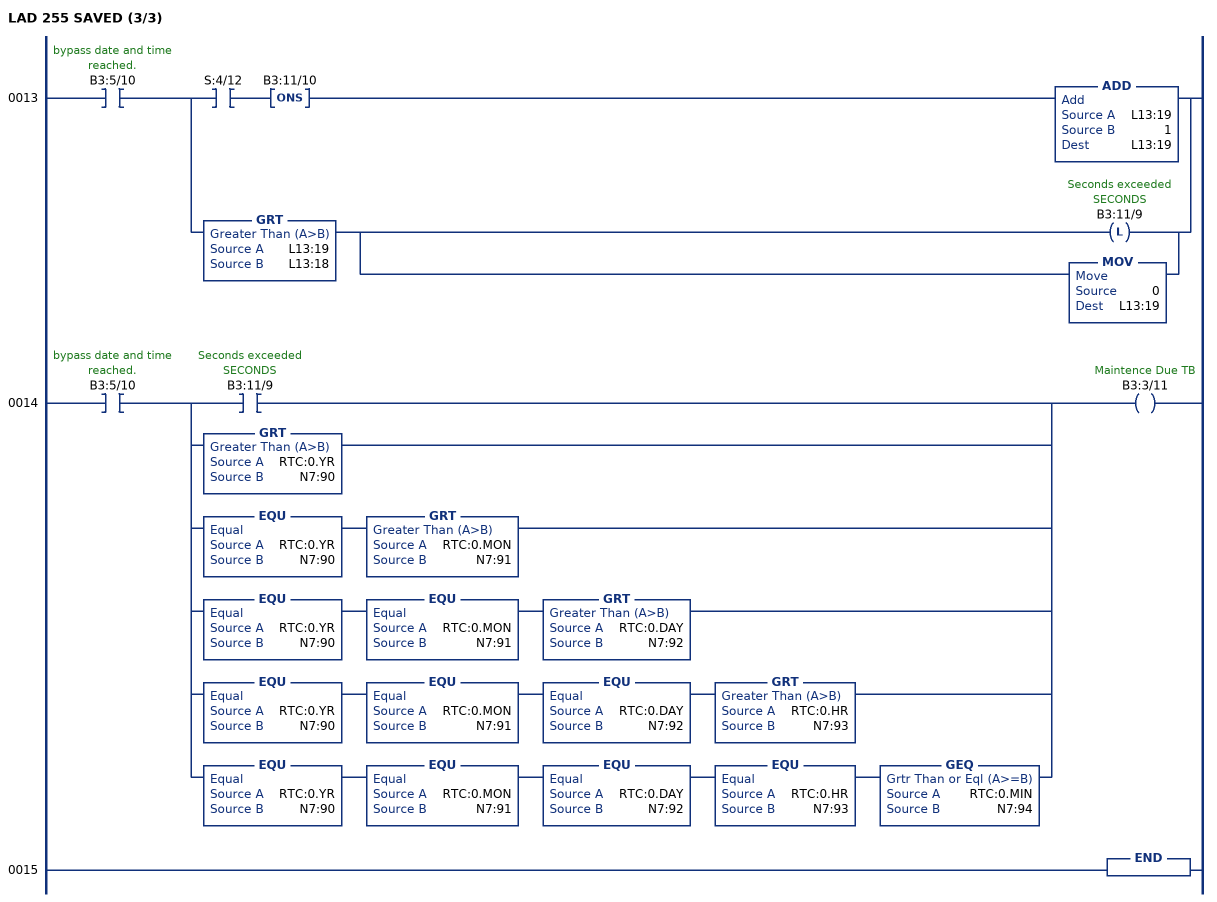
% Rung: 13 %
SOR XIC B3:5/10 BST XIC S:4/12 ONS B3:11/10 ADD L13:19 1 L13:19 NXB GRT L13:19 L13:18 BST OTL B3:11/9 NXB MOV 0 L13:19 BND BND EOR
%   B3:5/10  "bypass date and time reached." %
%   L13:18  MAX %
%   B3:11/9  SECONDS  "Seconds exceeded" %
% Rung: 14 %
SOR XIC B3:5/10 BST XIC B3:11/9 NXB GRT RTC:0.YR N7:90 NXB EQU RTC:0.YR N7:90 GRT RTC:0.MON N7:91 NXB EQU RTC:0.YR N7:90 EQU RTC:0.MON N7:91 GRT RTC:0.DAY N7:92 NXB EQU RTC:0.YR N7:90 EQU RTC:0.MON N7:91 EQU RTC:0.DAY N7:92 GRT RTC:0.HR N7:93 NXB EQU RTC:0.YR N7:90 EQU RTC:0.MON N7:91 EQU RTC:0.DAY N7:92 EQU RTC:0.HR N7:93 GEQ RTC:0.MIN N7:94 BND OTE B3:3/11 EOR
%   B3:5/10  "bypass date and time reached." %
%   B3:11/9  SECONDS  "Seconds exceeded" %
%   N7:90  RTC %
%   B3:3/11  TB  "Maintence Due" %
% Rung: 15 %
SOR END EOR

OTHER DOCUMENTED ADDRESSES
  B3:0/1  "toggle"
  B3:0/13  "toggle 2"
  B3:10/1  "bypass"
  B189:0/0  "change box"
  B189:0/9  "override boxing ok or not full signal"
  B189:0/11  "HMI force door close"
  B196:1/0  "Chute door is closed"
  B196:1/1  "control chute door"
  B196:1/13  "force box conveyor on"
  B196:3/0  "for hmi to continue production unlatched by hmi"
  HSC:0.0  "top"
  HSC:0.3/6  "Underflow interrupt"
  HSC:0.3/7  "Overflow interrupt"
  HSC:1.0  "bot"
  HSC:1.3/6  "Underflow interrupt"
  HSC:1.3/7  "Overflow interrupt"
  I:0.0/0  "Encoder Signal "A""
  I:0.0/1  "Encoder Signal "B""
  I:0.0/4  "Encoder Signal "A""
  I:0.0/5  "Encoder Signal "B""
  I:0.1/4  "not used"
  I:0.1/5  "not used"
  I:0.1/6  "not used"
  I:0.1/7  "not used"
  I:0.1/8  "not used"
  I:0.1/9  "not used"
  I:0.1/10  "not used"
  I:0.1/11  "not used"
  I:0.1/12  "not used"
  I:0.1/13  "not used"
  I:0.1/14  "not used"
  I:0.1/15  "not used"
  I:0.2  "not used"
  I:0.2/3  "Packaging Conveyor full"
  I:0.2/4  "Packaging Conveyor Box in Position"
  I:0.3  "not used"
  I:0.4  "Spare Analog Input 1"
  I:0.5  "Spare Analog Input 2"
  I:0.6  "Spare Analog Input 3"
  I:2.0/0  FRONT_ESTOP
  I:2.0/1  REAR_ESTOP
  I:2.0/8  FRONT_DOOR  "front door signal ce models only"
  I:2.0/9  REAR_DOOR  "rear door signal ce models only"
  I:2.0/11  "spare"
  L23:19  TOP_OPT_FAIL_CT
  L23:34  AIR_PRESSURE_FAULT
  L28:0  INS_1_TIME
  L29:0  INS_1_POS
  L30:0  INS_5_TIME
  L31:0  INS_5_POS
  L32:0  INS_6_TIME
  L33:0  INS_6_POS
  L192:1  BOT_LAST_TIME  "rtc bot belt previous movement event time"
  L192:2  BOT_CYCLE_TIME  "rtc bot belt time between events"
  L192:7  FROM_REAL  "distance from real part signal at optic location"
  L192:8  FROM_TRACKED  "distance from tracked part signal at optic location"
  L192:16  TOP_LAST_TIME  "rtc top belt previous movement event time"
  L192:17  TOP_CYCLE_TIME  "rtc top belt time between events"
  L199:5  ACQTM51
  L199:6  ACQTM52
  L199:7  ACQTM53
  L199:9  "ones"
  L199:10  "billions"
  L199:13  DUMP_LONG
  L199:15  ACQTM11
  L199:16  ACQTM12
  L199:17  ACQTM13
  L199:20  RESULTTM1
  L199:22  CLEARTIME5COUNT
  L199:23  CLEARTIME6COUNT
  L199:24  ACQTM61
  L199:25  ACQTM62
  L199:26  ACQTM63
  L199:27  TMSINCETRIG1
  L199:29  TMSINCETRIG5
  L199:30  TMSINCETRIG6
  L199:31  CLEARTIME1COUNT
  L199:32  RESULTTM5
  L199:33  RESULTTM6
  L199:34  MAXACQTM1
  L199:36  MAXACQTM6
  N7  
  N101:1  I2_TRIG_LOC
  N101:2  I3_TRIG_LOC
  N101:3  I4_TRIG_LOC
  O:0.0/1  "spare"
  O:0.0/11  "Spare"
  O:0.0/12  "not used"
  O:0.0/13  "not used"
  O:0.0/14  "not used"
  O:0.0/15  "not used"
  O:0.1  "not used"
  O:0.2  "not used"
  O:0.3  "not used"
  O:0.5  "spare analog output"
  O:3.0/0  "spare"
  O:3.0/2  "spare"
  O:3.0/3  "light curtain range selection /* needed? */"
  O:3.0/7  "door unlocks on CE models"
  O:3.0/8  "Light?"
  PFILE:6  "check for part jams"
  PFILE:10  "Bottom belt HSC"
  PFILE:12  "Top belt HSC"
  Q2:55  END_OF_MAIN
  Q5:94  END_OF_BELTS
  T20:0  "Trigger On Time"
  U:9  "slow data"
  U:24  "check skipped fail rate"
  U:28  "faults"
  U:29  "speed"
  U:30  "count"
  U:31  "rate calc"
  U:32  "boxer"
  U:33  "bulk pack"
  U:34  "customer boxing unit signals"
  U:35  "cleanup"

COMMENTS NOT ATTACHED TO A CURRENT RUNG
  R6:2: B41 is the top good 3 file
  R6:6/DN: B35 is the top NG file
  R6:10/DN: B37 is the top good 1 file
  R6:11/DN: B39 is the top good 2 file
  R6:0: B36 is the bottom GOOD file
  R6:10: B37 is the top good 1 file
  R6:6: B35 is the top NG file
  R6:4: B34 is the bottom NG file

REVISION NOTES
  13: updated count reset
  14: added io moduals
  15: multiple steps toward new hmi integration
  21: test
  27: fix error if bulk pack and no boxing fallout were on

DATA TABLE (non-zero values as saved)
DATA B3
% B3:0 % 0X8032 0X0341 0X4001 0X9109 0X0EF3 0X0534 0X0C80 0X0420 0X2F80 0X22B0
% B3:10 % 0X201C 0X00CE 0X4000 0X8000 0X0000 0X0000 0X0000 0X0000 0X0000 0X0000
% B3:50 % 0X0001 0X0000 0X0000 0X0000 0X0000 0X0000 0X0000 0X0000 0X0000 0X0000
DATA T4
% .PRE .ACC %
% T4:0 % 0 3
% T4:1 % 150 0
% T4:2 % 400 0
% T4:3 % 250 98
% T4:4 % 1000 0
% T4:5 % 5 5
% T4:6 % 10 10
% T4:7 % 150 0
% T4:8 % 20 5
% T4:9 % 50 35
% T4:10 % 200 200
% T4:11 % 111 0
% T4:12 % 20 24
% T4:13 % 250 0
% T4:14 % 666 0
% T4:15 % 1000 1000
% T4:16 % 400 0
% T4:17 % 100 90
% T4:18 % 5 0
% T4:19 % 300 0
% T4:20 % 200 0
% T4:21 % 200 0
% T4:22 % 200 0
% T4:23 % 250 0
% T4:24 % 666 0
% T4:25 % 666 0
% T4:26 % 666 0
% T4:27 % 250 0
% T4:28 % 250 0
% T4:29 % 5000 0
% T4:30 % 333 111
% T4:31 % 333 110
% T4:32 % 250 100
% T4:33 % 250 103
DATA C5
% .PRE .ACC %
% C5:0 % 32766 0
DATA R6
% .LEN .POS %
% R6:0 % 1250 0
% R6:1 % 16 0
% R6:2 % 1050 0
% R6:3 % 1050 0
% R6:4 % 1250 0
% R6:5 % 1250 0
% R6:6 % 1713 0
% R6:7 % 16 0
% R6:8 % 1024 0
% R6:9 % 3 0
% R6:10 % 1713 0
% R6:11 % 1050 0
% R6:12 % 10 0
% R6:13 % 10 0
% R6:14 % 10 0
% R6:15 % 10 0
% R6:16 % 1713 0
% R6:17 % 1713 0
% R6:18 % 1050 0
% R6:19 % 10 0
DATA N7
% N7:0 % 17247 3 1027 300 3 0 0 0 500 43
% N7:10 % 1000 43 0 2 20 20 1000 2000 50 1050
% N7:20 % 0 1329 10 2000 222 46 0 0 48 250
% N7:30 % 666 1418 150 0 0 1231 77 8 0 8
% N7:40 % 3 1 0 1 32767 482 1216 1350 1636 0
% N7:50 % 0 0 0 16 1 1024 0 0 32766 3
% N7:60 % 1713 1713 1050 984 1034 1024 4999 5 400 400
% N7:70 % 100 200 300 400 90 190 290 390 16428 15889
% N7:80 % 0 0 1238 1246 1300 1310 3 36 0 0
% N7:90 % 2011 4 4 12 1 3 36 222 222 12
% N7:100 % 1003 90 110 100 175 25 0 0 0 0
% N7:190 % -128 27477 27605 32767 0 0 0 0 0 0
DATA F8
% F8:0 % 6
DATA L13
% L13:0 % 12164 115601 0 35055 169076
% L13:5 % 131 4210 131 131393 111
% L13:10 % 111 96816498 30832 15 90
% L13:15 % 1573710681 -2147483648 2147483647 2147483647 82058
% L13:20 % 36582183 2059927638 777 33125 100
% L13:25 % 82 2232 91700508 111 1409426104
% L13:30 % 164283673 131 60000 1097515367 444
% L13:35 % 0 96 99 -301123785 -301123762
% L13:40 % 10303 1000000000 1000000 1097515339 1572623747
% L13:45 % 1572623775 23 0 28 3523382
% L13:50 % 1086934 67188061 1563376893 0 0
% L13:55 % 1086906 20455 7528 230 -1783954972
% L13:60 % 26 104 -1783954986 600 0
% L13:65 % 100 0 -301150540 -301150945 12
% L13:70 % 2057842783 8 118 1030300 3523382
% L13:75 % 8919967 60 100 1563376901 13
% L13:80 % 24 74 962 7 752804
% L13:85 % 39418253 100 102 0 1086935
% L13:90 % 1086907 5 34857 5 1572623773
% L13:95 % 10 228 0 1572623798 89410
% L13:100 % 2147483647 6 900 14 508
% L13:105 % 89410 31 2099392 4691 2099386
% L13:110 % 6 100 50 1923692887 2020509362
% L13:115 % 2020509385 23 12 2020509373 26
% L13:120 % 4 5845 50 100 10
% L13:125 % 0 2057842783 2147483647 3276500 136234751
% L13:130 % 2 2 0 99 0
% L13:135 % 0 0 39418253 5 70
% L13:140 % 0 5 36 50 50
% L13:145 % 67188168 5 5 5 8
% L13:150 % 12 20 5115990 -5115990 96816498
% L13:155 % 0 -10 0 0 4589052
% L13:160 % 6 26 23 1220 45
% L13:165 % 2059708501 2059708507 2059708501 2059708507 6706
% L13:170 % 12817 254 255 1200 700
% L13:175 % 4 4 42 23 38
% L13:180 % -301114591 72 51008 1000000 102000000
% L13:185 % 0 0 -301114510 73 50325
% L13:190 % 100000000 0 0 0 0
DATA L19
% L19:0 % 1409426104 1409431911 1409437126 1409442330 1409448715
% L19:5 % 1409455142 1409462880 1409468857 1409350917 1409354638
% L19:10 % 1409358086 1409390096 1409395287 1409401188 1409407615
% L19:15 % 1409413759 1409420249 0 0 0
DATA L20
% L20:0 % 1572621964 1572623239 1572623493 1572623747 1562506356
% L20:5 % 1562506610 1562507882 1562508137 1562508392 1562549323
% L20:10 % 1562550840 1562854294 1562854549 1562855822 1562856076
% L20:15 % 1562856331 1562888045 1562889564 1562890069 1563063132
% L20:20 % 1563063387 1563064659 1563064914 1563065169 1563288929
% L20:25 % 1563290446 1563325836 1563326090 1563327362 1563327616
% L20:30 % 1563327871 1563374911 1563376426 1563376934 1563405555
% L20:35 % 1563405808 1563407081 1563407335 1563407589 1563717067
% L20:40 % 1563717323 1563718595 1563718849 1563719104 1568539702
% L20:45 % 1568539956 1568541229 1568541484 1568541737 1572621710
DATA L21
% L21:0 % 2059708143 2059708399 2059708450 2059708501 2057641092
% L21:5 % 2057641153 2057641439 2057641493 2057641547 2057649801
% L21:10 % 2057650149 2057726611 2057726671 2057726950 2057727004
% L21:15 % 2057727056 2057733453 2057733805 2057733928 2057777542
% L21:20 % 2057777603 2057777889 2057777943 2057777997 2057823112
% L21:25 % 2057823465 2057832381 2057832442 2057832731 2057832785
% L21:30 % 2057832839 2057842325 2057842669 2057842793 2057850006
% L21:35 % 2057850067 2057850355 2057850409 2057850463 2057912852
% L21:40 % 2057912904 2057913160 2057913211 2057913263 2058885124
% L21:45 % 2058885175 2058885432 2058885483 2058885534 2059708091
DATA L22
% L22:0 % 1562890103 1563063162 1563063418 1563064689 1563064943
% L22:5 % 1563065197 1563288989 1563290503 1563291008 1563325866
% L22:10 % 1563326121 1563327396 1563327650 1563327904 1563374950
% L22:15 % 1563376465 1563376972 1563405586 1563405841 1563407112
% L22:20 % 1563407366 1563407621 1563717105 1563717358 1563718629
% L22:25 % 1563718884 1563719139 1568539729 1568539984 1568541255
% L22:30 % 1568541509 1568541764 1572621743 1572621995 1572623266
% L22:35 % 1572623520 1572623775 1562507910 1562508164 1562508419
% L22:40 % 1562549352 1562550867 1562551373 1562854324 1562854576
% L22:45 % 1562855850 1562856103 1562856357 1562888081 1562889597
DATA L23
% L23:0 % 2057733937 2057777549 2057777610 2057777895 2057777949
% L23:5 % 2057778002 2057823125 2057823479 2057823603 2057832388
% L23:10 % 2057832449 2057832738 2057832792 2057832846 2057842334
% L23:15 % 2057842679 2057842802 2057850014 2057850075 2057850362
% L23:20 % 2057850416 2057850469 2057912860 2057912911 2057913167
% L23:25 % 2057913218 2057913270 2058885129 2058885181 2058885437
% L23:30 % 2058885488 2058885540 2059708098 2059708149 2059708405
% L23:35 % 2059708456 2059708507 2057641445 2057641499 2057641553
% L23:40 % 2057649808 2057650155 2057650278 2057726618 2057726677
% L23:45 % 2057726956 2057727009 2057727062 2057733461 2057733813
DATA L30
% L30:0 % 1097513510 1097513738 1097513967 1097514196 1097514426
% L30:5 % 1097514655 1097514883 1097515111 1097515339 1071304727
% L30:10 % 1071304952 1071305179 1071305406 1071305631 1071305859
% L30:15 % 1071306086 1071306312 1071306539 1071306765 1071306992
% L30:20 % 1071307217 1071307442 1071307668 1071307895 1071308121
% L30:25 % 1071308347 1071308573 1071308799 1071309024 1071309250
% L30:30 % 1071309476 1071429569 1071429795 1071431153 1071431379
% L30:35 % 1071431606 1088333039 1088333266 1088334623 1088334848
% L30:40 % 1088335075 1089808842 1089809070 1089810430 1089810657
% L30:45 % 1089810882 1092780028 1092791426 1092806921 1097513283
DATA L31
% L31:0 % 3522828 3522897 3522967 3523035 3523105
% L31:5 % 3523175 3523244 3523313 3523382 2077757
% L31:10 % 2077757 2077757 2077757 2077757 2077757
% L31:15 % 2077757 2077757 2077757 2077757 2077757
% L31:20 % 2077757 2077757 2077757 2077757 2077757
% L31:25 % 2077757 2077757 2077757 2077757 2077757
% L31:30 % 2077757 2077757 2077757 2077757 2077757
% L31:35 % 2077757 2077757 2077757 2077757 2077757
% L31:40 % 2077757 2077757 2077757 2077757 2077757
% L31:45 % 2077757 2091375 2094821 2099507 3522760
DATA L32
% L32:0 % 1563376385 1563376893 1409358274 1409390283 1409395476
% L32:5 % 1409401377 1409407804 1409413948 1409420437 1409426296
% L32:10 % 1409432104 1409437319 1409442521 1409448908 1409455334
% L32:15 % 1409463068 1409469047 1485322487 1485324003 1486084839
% L32:20 % 1486085343 1486085850 1486086357 1486086862 1486200075
% L32:25 % 1486201593 1486202099 1486227449 1486227954 1486228459
% L32:30 % 1486228965 1486229470 1562314458 1562317108 1562318624
% L32:35 % 1562319131 1562546873 1562549286 1562550803 1562551308
% L32:40 % 1562885434 1562888017 1562889533 1562890041 1563286489
% L32:45 % 1563288874 1563290389 1563290894 1563372344 1563374872
DATA L33
% L33:0 % 2057842660 2057842783 2020401255 2020432555 2020437631
% L33:5 % 2020443402 2020449688 2020455695 2020462040 2020467771
% L33:10 % 2020473451 2020478550 2020483638 2020489883 2020496169
% L33:15 % 2020503729 2020509574 2042023076 2042023535 2042215265
% L33:20 % 2042215393 2042215520 2042215648 2042215775 2042244305
% L33:25 % 2042244689 2042244816 2042251204 2042251331 2042251459
% L33:30 % 2042251586 2042251714 2057592897 2057593437 2057593787
% L33:35 % 2057593911 2057649303 2057649793 2057650140 2057650262
% L33:40 % 2057732919 2057733447 2057733797 2057733921 2057822611
% L33:45 % 2057823100 2057823451 2057823574 2057841803 2057842317
DATA B40
% B40:0 % 0XAAAA
DATA B100
% B100:0 % 0X2780 0X18A0 0X0004 0X0000 0X0000 0X0000 0X0000 0X0000 0X0000 0X0000
DATA N101
% N101:0 % 118 0 0 0 1183 100 1002 1200 1212 1230
% N101:10 % 1240 1604 10 16383 1269 17365 2974 250 333 333
% N101:20 % 1000 500 400 0 0 0 250 250 0 0
DATA L102
% L102:0 % 20 10 2000 1987 2000
% L102:5 % 2000 0 0 0 0
% L102:10 % 0 115 0 0 34857
% L102:15 % 0 30 10 30 10
% L102:20 % 0 12 67755 5 26
% L102:25 % 28 0 66252844 81649 9418788
% L102:30 % 8 0 9 7746 2
% L102:35 % 174 302 0 999999 23
% L102:40 % 1 7 63154 3 0
